// TIA Portal V17 export
// export: Created 2022-01-24T16:52:05.0564952Z, ExportSetting WithDefaults, DisplayName Totally Integrated Automation Portal, DisplayVersion V17, DisplayName TIA Portal Openness, DisplayVersion V17, DisplayName TIA Portal Version Control Interface, DisplayVersion V17, DisplayName SINAMICS Startdrive Advanced, DisplayVersion V17, DisplayName SINAMICS Startdrive G130, G150, S120, S150, SINAMICS MV, S210, DisplayVersion V17, DisplayName SINAMICS Startdrive G110M, G120, G120C, G120D, G120P, G115D, DisplayVersion V17, DisplayName STEP 7 Professional, DisplayVersion V17, DisplayName STEP 7 Safety, DisplayVersion V17, DisplayName WinCC Advanced, DisplayVersion V17
FUNCTION_BLOCK "funkce2"   // FB1, LAD
{ S7_Optimized_Access := 'TRUE' }
VERSION : 0.1
// stored: AutoNumber true, IsIECCheckEnabled false, IsRetainMemResEnabled false, MemoryReserve 100, SetENOAutomatically false, UDAEnableTagReadback false
   VAR_INPUT
      start : Bool;
      stop : Bool;
   END_VAR
   VAR_OUTPUT
      motorBeh : Bool;
   END_VAR
   VAR
      statMotorBeh : Bool;
   END_VAR
   VAR_TEMP   // added for the SCL form of the ladder/FBD networks
      _w1 : Bool;
   END_VAR
BEGIN

REGION Network 1
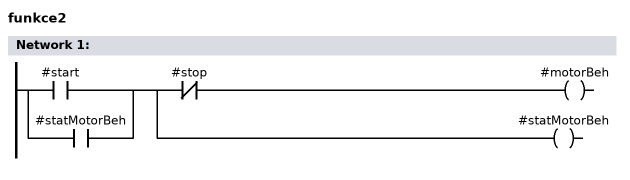
   RUNG wire#powerrail
      Contact( #start )
      wire#w1
      I_Contact( #stop )
      Coil( #motorBeh )
   END_RUNG
   RUNG wire#powerrail
      Contact( #statMotorBeh )
   END_RUNG wire#w1
   RUNG wire#w1
      Coil( #statMotorBeh )
   END_RUNG
   // the same network as SCL:
   #_w1 := #start OR #statMotorBeh;
   #motorBeh := #_w1 AND NOT #stop;
   #statMotorBeh := #_w1;
END_REGION
END_FUNCTION_BLOCK
